TYPE CoverPanelSetStatuses :
STRUCT
	apertureStatus: ApertureStatus;
	healthStatus: HealthStatus;
	busyStatus: BusyStatus;
END_STRUCT
END_TYPE

(* stored: Version 1.1.0.1, ProductVersion 3.1.4019.2
   DUT CoverPanelSetStatuses: Id {f44f98de-f3ad-479c-87a4-8949da8599fe} *)
